(* PLC project  *)

CONFIGURATION VirtualBox
END_CONFIGURATION
